(*
Adds a fixed offset to the input signal.

A positive value shifts the output up; a negative value shifts it down.
*)
{attribute 'enable_dynamic_creation'}
{attribute 'no_explicit_call' := 'direct call for this function block is not allowed'}
FUNCTION_BLOCK FINAL FB_Bias EXTENDS FB_SisoComponent
IMPLEMENTS FsCommon.I_Runnable
VAR
	_fBias : LREAL; // Fixed offset added to the input.
END_VAR

(* Gets or sets the fixed offset added to the input. Negative values subtract. *)
PROPERTY Bias : LREAL
GET
Bias := THIS^._fBias;
END_GET
SET
THIS^._fBias := Bias;
END_SET
END_PROPERTY

METHOD FB_init : BOOL
VAR_INPUT
	bInitRetains : BOOL; // if TRUE, the retain variables are initialized (warm start / cold start)
	bInCopyCode  : BOOL;  // if TRUE, the instance afterwards gets moved into the copy code (online change)
	fBias        : LREAL; // Fixed offset added to the input.
END_VAR
THIS^._fBias := fBias;
END_METHOD

(* Adds :attr:`Bias` to the current input. *)
METHOD Run
VAR_INPUT
END_VAR
THIS^._fOutput := THIS^._fInput + THIS^._fBias;
END_METHOD

END_FUNCTION_BLOCK

(* stored: Version 1.1.0.1, ProductVersion 3.1.4024.15
   POU FB_Bias: Id {49e29d60-f729-0376-0c75-4ceaf1c6c44d}, SpecialFunc None
   Property Bias: Id {8ba14310-58ed-0393-2100-54f7aa4ae283}
   Get Get: Id {7cae08ca-54d3-0f6f-04ba-658962e49d8f}
   Set Set: Id {21546a0d-21b8-0c03-2d7d-a29be2bd0584}
   Method FB_init: Id {d6080596-1986-001a-3232-78b3ef086d35}
   Method Run: Id {91912f97-af7b-0653-2a68-d5157071b51d} *)
